(* PLC project Senza_nome, Sconosciuto Senza_nome 1 *)
(* stored: creationDateTime 2020-04-13T10:39:50, modificationDateTime 2020-06-24T12:04:16 *)

FUNCTION_BLOCK genera
  VAR_INPUT
    generate : BOOL;  (* generazione di un nuovo veicolo all'ingresso *)
  END_VAR
  VAR
    veicoli : ARRAY[1..10] OF INT;
    current_array_pos : INT := 1;
  END_VAR
  VAR_OUTPUT
    weight : INT;  (* peso "rilevato" *)
  END_VAR

            (* Blocco che simula l'ingresso di veicoli di differente peso*)
(* peso<=250= moto, peso>250 & peso <900= auto, peso>=900=camion*)

(* Definizione valori array di prova*)
veicoli[1] := 100;
veicoli[2] := 1454;
veicoli[3] := 807;
veicoli[4] := 252;
veicoli[5] := 1068;
veicoli[6] := 908;
veicoli[7] := 309;
veicoli[8] := 154;
veicoli[9] := 603;
veicoli[10] := 414;

if (generate=TRUE) then
  weight := veicoli[current_array_pos];
end_if;

current_array_pos := current_array_pos + 1;

(* Evito overflow array*)
if current_array_pos > 10 then
  current_array_pos := 1;
end_if;



          
END_FUNCTION_BLOCK

FUNCTION_BLOCK exit_sel
  VAR_INPUT
    confirm : BOOL := 0;  (* conferma veicolo in uscita *)
    slct : BOOL := 0;  (* selezione veicolo in uscita *)
  END_VAR
  VAR_OUTPUT
    veicolo : REAL;  (* veicolo selezionato *)
  END_VAR
  VAR
    auto : REAL := 1.0;
    moto : REAL := 0.50;
    camion : REAL := 2.0;
  END_VAR
  VAR_OUTPUT
    apri_sbarra : BOOL := 0;  (* abilitazione della sbarra d'uscita al piano *)
    cat : STRING;  (* uscita a monitor del tipo di veicolo in uscita *)
  END_VAR
  VAR
    tipo : INT;  (* tipologia di veicolo in uscita *)
    R_TRIG0 : R_TRIG;
  END_VAR

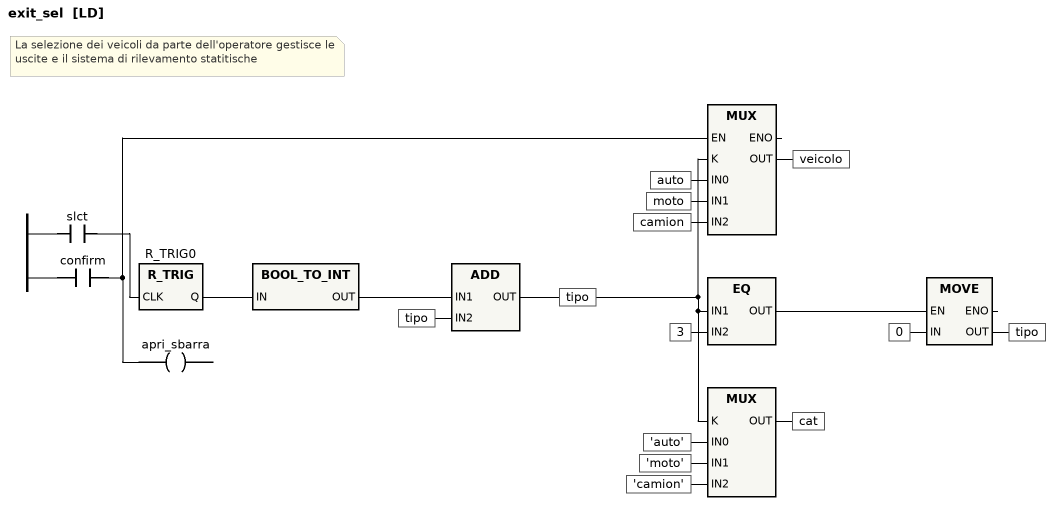
(* LD diagram, written out as Structured Text *)
IF confirm THEN veicolo := MUX(tipo, auto, moto, camion); END_IF;
apri_sbarra := confirm;
R_TRIG0(CLK := slct);
tipo := BOOL_TO_INT(R_TRIG0.Q) + tipo;
cat := MUX(tipo, 'auto', 'moto', 'camion');
(* La selezione dei veicoli da parte dell'operatore gestisce le uscite e il sistema di rilevamento statitische *)
IF tipo = 3 THEN tipo := 0; END_IF;
END_FUNCTION_BLOCK

FUNCTION_BLOCK gettoniera
  VAR_INPUT
    enable : BOOL := 0;  (* abilitazione/disabilitazione pagamento *)
    euro_1 : BOOL := 0;  (* rileva l'inserimento di 1€ *)
    euro_2 : BOOL := 0;  (* rileva l'inserimento di 2€ *)
    euro_50c : BOOL := 0;  (* rileva l'inserimento di 0.50€ *)
    ore : BOOL := 0;  (* ore di permanenza nel parcheggio *)
    tariffa : REAL := 1.0;  (* tariffa applicata in base al tipo di veicolo *)
  END_VAR
  VAR
    tot : REAL := 0.0;  (* totale inserito dall'utente *)
    prc : REAL := 1.0;
  END_VAR
  VAR_OUTPUT
    prezzo : REAL := 1.0;  (* uscita a schermo prezzo parcheggio *)
    tot_mon : REAL := 0.0;  (* uscita a schermo totale inserito *)
    hrs : INT := 0;  (* uscita a schermo ore *)
  END_VAR
  VAR
    ora : INT := 1;  (* conteggio delle ore *)
  END_VAR
  VAR_OUTPUT
    apri_sbarra : BOOL := 0;  (* apertura della sbarra dopo il pagamento *)
  END_VAR
  VAR
    R_TRIG0 : R_TRIG;
    R_TRIG1 : R_TRIG;
  END_VAR
  VAR_OUTPUT
    resto : REAL := 0.0;  (* resto erogato *)
  END_VAR
  VAR
    R_TRIG2 : R_TRIG;
    R_TRIG3 : R_TRIG;
    R_TRIG4 : R_TRIG;
    CTUD0 : CTUD;
  END_VAR
  VAR  (* added by the conversion: wires and edge detectors of the diagram *)
    R_TRIG1_2 : R_TRIG;
    _ADD185_OUT : REAL;
    _GE14_ENO : BOOL;
    _GE14_OUT : BOOL;
    R_TRIG2_2 : R_TRIG;
    _ADD16_ENO : BOOL;
    _ADD16_OUT : REAL;
    R_TRIG3_2 : R_TRIG;
    _SUB171_ENO : BOOL;
    _SUB171_OUT : REAL;
    _MOVE134_ENO : BOOL;
    _MOVE134_OUT : REAL;
    _LIMIT200_OUT : INT;
    _BOOL_TO_INT161_ENO : BOOL;
    _BOOL_TO_INT161_OUT : INT;
  END_VAR

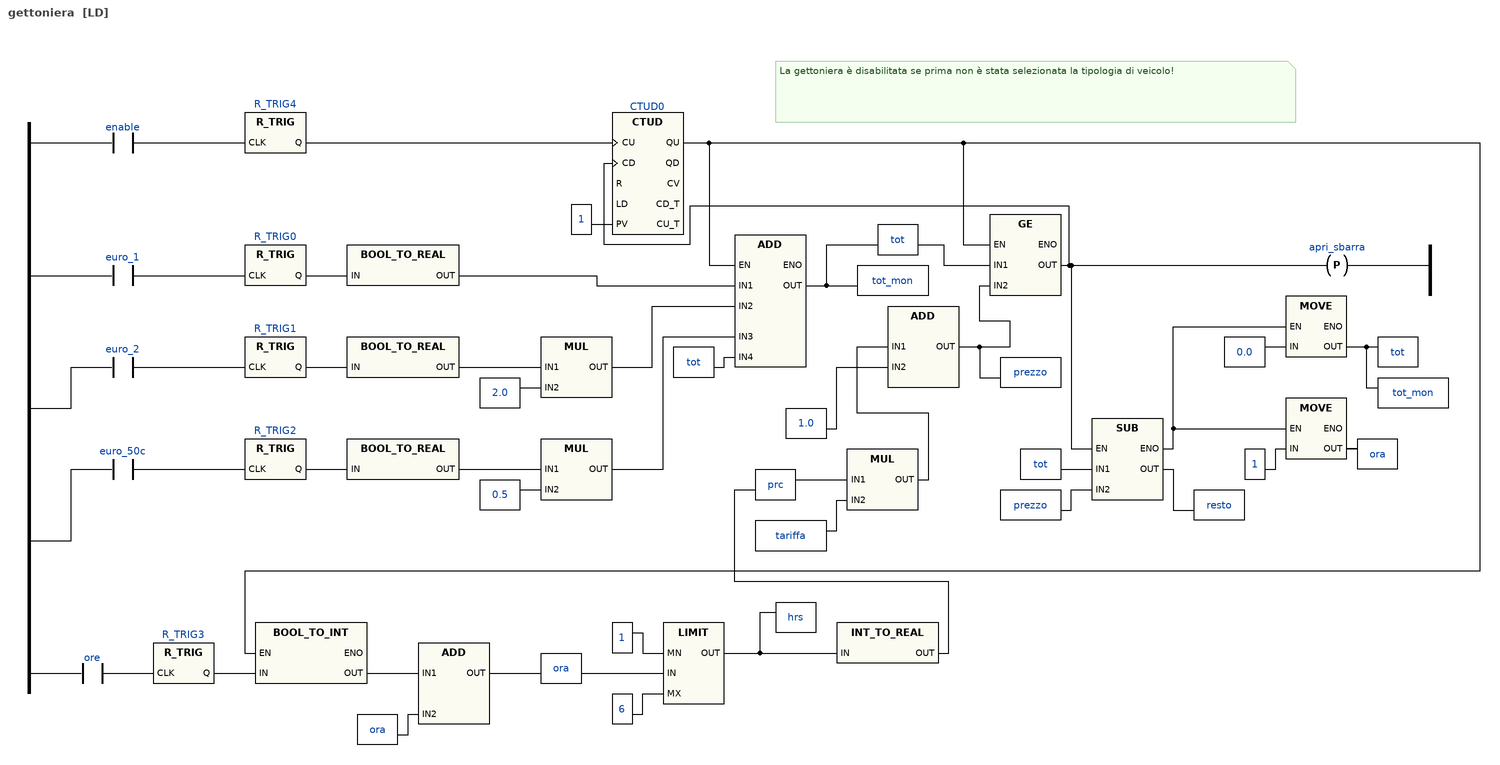
(* LD diagram, written out as Structured Text *)
(* La gettoniera è disabilitata se prima non è stata selezionata la tipologia di veicolo! *)
R_TRIG4(CLK := enable);
R_TRIG1_2(CLK := R_TRIG4.Q);
_ADD185_OUT := prc * tariffa + 1.0;
_GE14_OUT := GE(EN := CTUD0.QU, IN1 := tot, IN2 := _ADD185_OUT, ENO => _GE14_ENO);
R_TRIG2_2(CLK := _GE14_OUT);
CTUD0(CU := R_TRIG1_2.Q, CD := R_TRIG2_2.Q, PV := 1);
R_TRIG0(CLK := euro_1);
R_TRIG1(CLK := euro_2);
R_TRIG2(CLK := euro_50c);
_ADD16_OUT := ADD(EN := CTUD0.QU, IN1 := BOOL_TO_REAL(R_TRIG0.Q), IN2 := BOOL_TO_REAL(R_TRIG1.Q) * 2.0, IN3 := BOOL_TO_REAL(R_TRIG2.Q) * 0.5, IN4 := tot, ENO => _ADD16_ENO);
IF _ADD16_ENO THEN tot := _ADD16_OUT; END_IF;
R_TRIG3_2(CLK := _GE14_OUT);
apri_sbarra := R_TRIG3_2.Q;
IF _ADD16_ENO THEN tot_mon := _ADD16_OUT; END_IF;
_SUB171_OUT := SUB(EN := _GE14_OUT, IN1 := tot, IN2 := prezzo, ENO => _SUB171_ENO);
_MOVE134_OUT := MOVE(EN := _SUB171_ENO, IN := 0.0, ENO => _MOVE134_ENO);
IF _MOVE134_ENO THEN tot := _MOVE134_OUT; END_IF;
prezzo := _ADD185_OUT;
IF _MOVE134_ENO THEN tot_mon := _MOVE134_OUT; END_IF;
IF _SUB171_ENO THEN ora := 1; END_IF;
_LIMIT200_OUT := LIMIT(1, ora, 6);
prc := INT_TO_REAL(_LIMIT200_OUT);
IF _SUB171_ENO THEN resto := _SUB171_OUT; END_IF;
hrs := _LIMIT200_OUT;
R_TRIG3(CLK := ore);
_BOOL_TO_INT161_OUT := BOOL_TO_INT(EN := CTUD0.QU, IN := R_TRIG3.Q, ENO => _BOOL_TO_INT161_ENO);
ora := _BOOL_TO_INT161_OUT + ora;
END_FUNCTION_BLOCK

FUNCTION_BLOCK park_stats
  VAR_INPUT
    en_calc : BOOL := 0;  (* abilitazione del conteggio dei ricavi *)
    guad : REAL;  (* pedaggio riscosso *)
    tot_auto1 : INT;  (* totale auto presenti piano terra *)
    tot_moto1 : INT;  (* totale moto presenti piano terra *)
    tot_camion1 : INT;  (* totale camion presenti piano terra *)
    tot_auto2 : INT;  (* totale auto presenti primo piano *)
    tot_moto2 : INT;  (* totale moto presenti primo piano *)
    tot_camion2 : INT;  (* totale camion presenti primo piano *)
  END_VAR
  VAR_OUTPUT
    tot_auto : INT := 0;  (* auto presenti nell'intero parcheggio *)
    tot_moto : INT := 0;  (* moto presenti nell'intero parcheggio *)
    tot_camion : INT := 0;  (* camion presenti nell'intero parcheggio *)
    incasso : REAL := 0.0;  (* incasso giornaliero *)
    daily_vhcl : INT := 0;  (* totale dei veicoli che hanno transitato in un giorno *)
  END_VAR
  VAR
    R_TRIG0 : R_TRIG;
  END_VAR

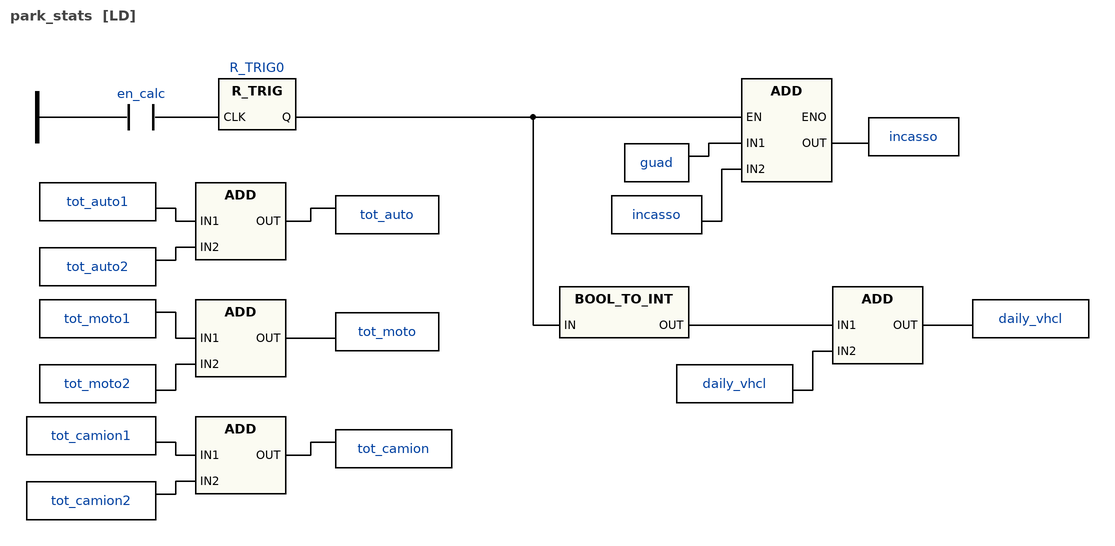
(* LD diagram, written out as Structured Text *)
R_TRIG0(CLK := en_calc);
IF R_TRIG0.Q THEN incasso := guad + incasso; END_IF;
tot_auto := tot_auto1 + tot_auto2;
daily_vhcl := BOOL_TO_INT(R_TRIG0.Q) + daily_vhcl;
tot_moto := tot_moto1 + tot_moto2;
tot_camion := tot_camion1 + tot_camion2;
END_FUNCTION_BLOCK

FUNCTION_BLOCK vehicle_cnt
  VAR_INPUT
    confirm_enter : BOOL := 0;  (* abilitazione per i contatori di incremento per un tipo di veicolo *)
    confirm_exit : BOOL := 0;  (* abilitazione per i contatori di decremento per un tipo di veicolo *)
    veicolo_in : REAL;  (* tipologia di veicolo in ingresso *)
    veicolo_out : REAL;  (* tipologia di veicolo in uscita *)
  END_VAR
  VAR_OUTPUT
    tot_auto : INT := 0;  (* totale auto presenti nel piano *)
    tot_moto : INT := 0;  (* totale moto presenti nel piano *)
    tot_camion : INT := 0;  (* totale camion presenti nel piano *)
  END_VAR
  VAR
    cap : INT := 4;  (* capacità di conteggio (legata al numero di veicoli per piano) *)
    R_TRIG0 : R_TRIG;
    CTUD0 : CTUD;
    CTUD1 : CTUD;
    CTUD2 : CTUD;
    R_TRIG1 : R_TRIG;
  END_VAR
  VAR  (* added by the conversion: wires and edge detectors of the diagram *)
    _EQ13_ENO : BOOL;
    _EQ13_OUT : BOOL;
    R_TRIG1_2 : R_TRIG;
    _EQ26_ENO : BOOL;
    _EQ26_OUT : BOOL;
    R_TRIG2 : R_TRIG;
    _EQ10_ENO : BOOL;
    _EQ10_OUT : BOOL;
    R_TRIG3 : R_TRIG;
    _EQ23_ENO : BOOL;
    _EQ23_OUT : BOOL;
    R_TRIG4 : R_TRIG;
    _EQ14_ENO : BOOL;
    _EQ14_OUT : BOOL;
    R_TRIG5 : R_TRIG;
    _EQ27_ENO : BOOL;
    _EQ27_OUT : BOOL;
    R_TRIG6 : R_TRIG;
  END_VAR

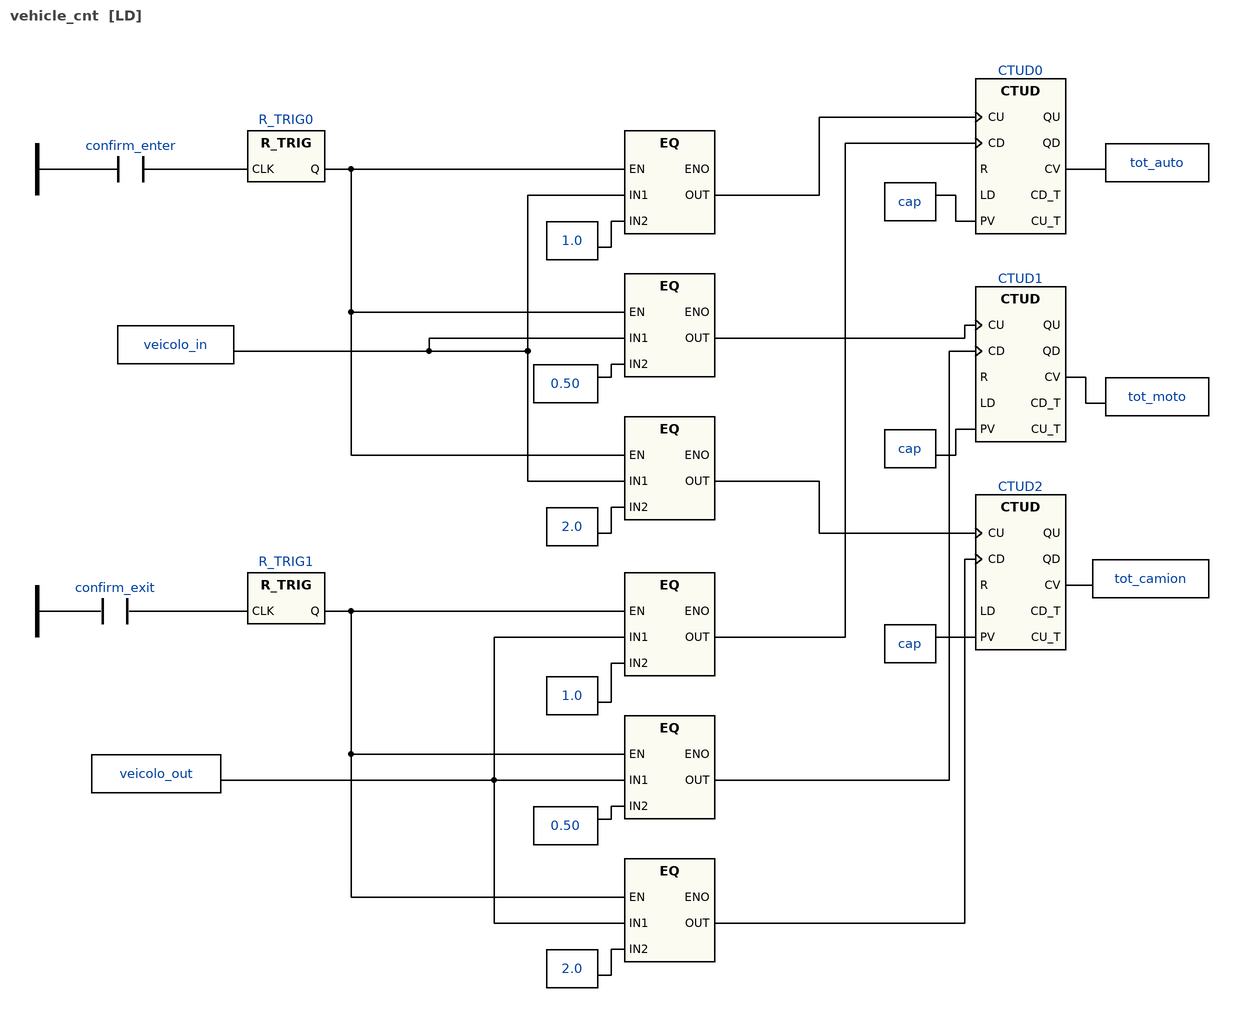
(* LD diagram, written out as Structured Text *)
R_TRIG0(CLK := confirm_enter);
_EQ13_OUT := EQ(EN := R_TRIG0.Q, IN1 := veicolo_in, IN2 := 1.0, ENO => _EQ13_ENO);
R_TRIG1_2(CLK := _EQ13_OUT);
R_TRIG1(CLK := confirm_exit);
_EQ26_OUT := EQ(EN := R_TRIG1.Q, IN1 := veicolo_out, IN2 := 1.0, ENO => _EQ26_ENO);
R_TRIG2(CLK := _EQ26_OUT);
CTUD0(CU := R_TRIG1_2.Q, CD := R_TRIG2.Q, PV := cap);
tot_auto := CTUD0.CV;
_EQ10_OUT := EQ(EN := R_TRIG0.Q, IN1 := veicolo_in, IN2 := 0.50, ENO => _EQ10_ENO);
R_TRIG3(CLK := _EQ10_OUT);
_EQ23_OUT := EQ(EN := R_TRIG1.Q, IN1 := veicolo_out, IN2 := 0.50, ENO => _EQ23_ENO);
R_TRIG4(CLK := _EQ23_OUT);
CTUD1(CU := R_TRIG3.Q, CD := R_TRIG4.Q, PV := cap);
tot_moto := CTUD1.CV;
_EQ14_OUT := EQ(EN := R_TRIG0.Q, IN1 := veicolo_in, IN2 := 2.0, ENO => _EQ14_ENO);
R_TRIG5(CLK := _EQ14_OUT);
_EQ27_OUT := EQ(EN := R_TRIG1.Q, IN1 := veicolo_out, IN2 := 2.0, ENO => _EQ27_ENO);
R_TRIG6(CLK := _EQ27_OUT);
CTUD2(CU := R_TRIG5.Q, CD := R_TRIG6.Q, PV := cap);
tot_camion := CTUD2.CV;
END_FUNCTION_BLOCK

FUNCTION_BLOCK vehicle_sel
  VAR_INPUT
    invio : BOOL := 0;  (* conferma scelta *)
    slct : BOOL := 0;  (* selezionatore (se >2 torna a 0) *)
    weight : INT;  (* rilevatore del peso del veicolo in ingresso *)
  END_VAR
  VAR_OUTPUT
    abilita : BOOL;  (* abilitazione gettoniera *)
    cat : STRING;  (* uscita a schermo *)
  END_VAR
  VAR
    veicleDetect : INT;  (* veicolo determinato in base al peso *)
  END_VAR
  VAR_OUTPUT
    veicolo : REAL := 1.0;  (* veicolo selezionato *)
  END_VAR
  VAR
    tipo : INT := 0;  (* auto=0, moto=1,camion=2 *)
    auto : REAL := 1.0;  (* tariffa auto *)
    moto : REAL := 0.50;  (* tariffa moto *)
    camion : REAL := 2.00;  (* tariffa camion *)
    R_TRIG0 : R_TRIG;
  END_VAR
  VAR  (* added by the conversion: wires and edge detectors of the diagram *)
    _AND61_OUT : BOOL;
    _AND44_OUT : BOOL;
    _GT47_OUT : BOOL;
    _EQ56_ENO : BOOL;
    _EQ56_OUT : BOOL;
    _MUX1_ENO : BOOL;
    _MUX1_OUT : REAL;
  END_VAR

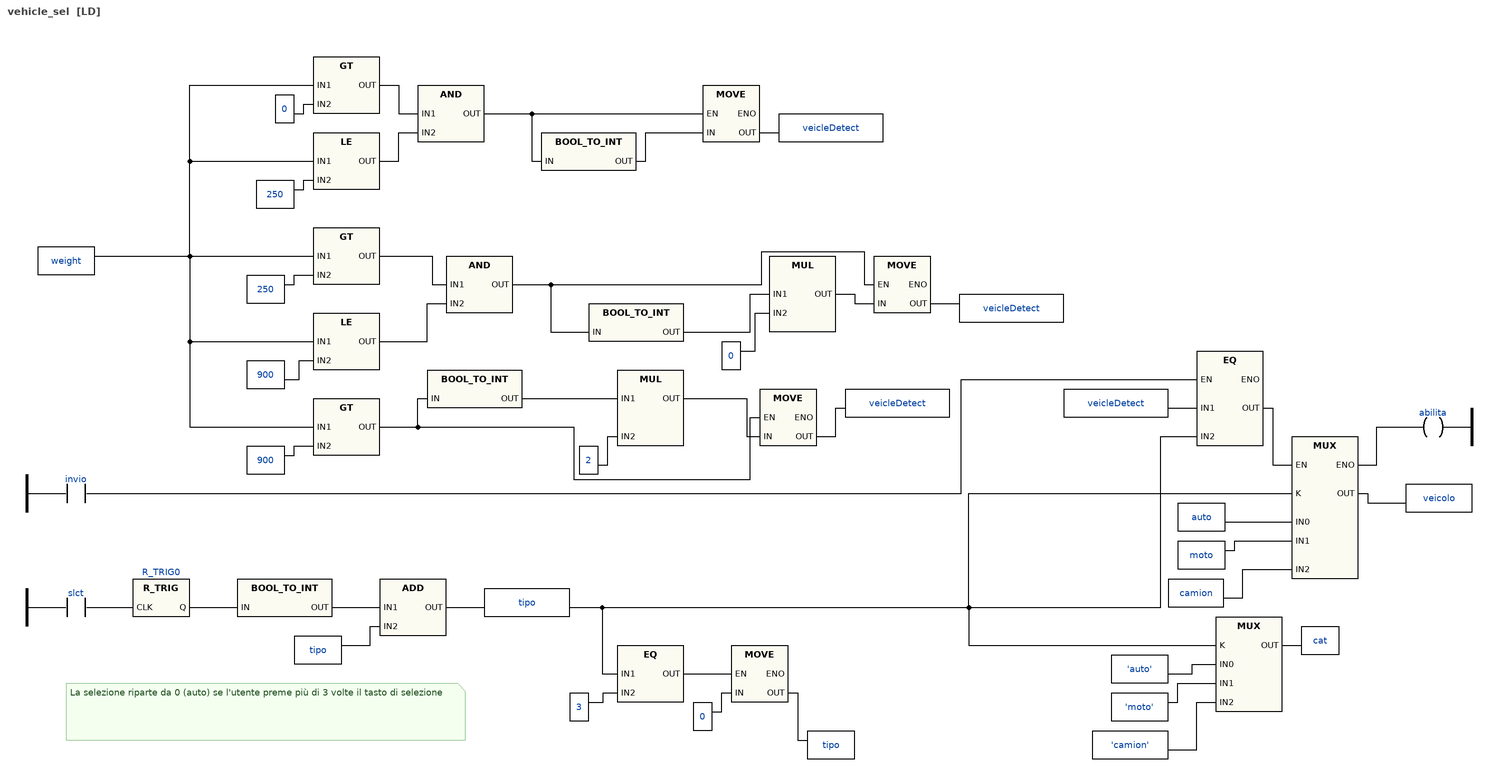
(* LD diagram, written out as Structured Text *)
_AND61_OUT := weight > 0 AND weight <= 250;
IF _AND61_OUT THEN veicleDetect := BOOL_TO_INT(_AND61_OUT); END_IF;
_AND44_OUT := weight > 250 AND weight <= 900;
IF _AND44_OUT THEN veicleDetect := BOOL_TO_INT(_AND44_OUT) * 0; END_IF;
_GT47_OUT := weight > 900;
IF _GT47_OUT THEN veicleDetect := BOOL_TO_INT(_GT47_OUT) * 2; END_IF;
_EQ56_OUT := EQ(EN := invio, IN1 := veicleDetect, IN2 := tipo, ENO => _EQ56_ENO);
_MUX1_OUT := MUX(EN := _EQ56_OUT, K := tipo, IN0 := auto, IN1 := moto, IN2 := camion, ENO => _MUX1_ENO);
abilita := _MUX1_ENO;
IF _MUX1_ENO THEN veicolo := _MUX1_OUT; END_IF;
R_TRIG0(CLK := slct);
tipo := BOOL_TO_INT(R_TRIG0.Q) + tipo;
cat := MUX(tipo, 'auto', 'moto', 'camion');
(* La selezione riparte da 0 (auto) se l'utente preme più di 3 volte il tasto di selezione *)
IF tipo = 3 THEN tipo := 0; END_IF;
END_FUNCTION_BLOCK

PROGRAM parking
  VAR
    start : BOOL := 0;  (* inizializzazione parcheggio *)
  END_VAR
  VAR_INPUT
    gen : BOOL := 0;  (* generazione veicolo *)
  END_VAR
  VAR
    slct : BOOL := 0;  (* selezione del tipo di veicolo (0 auto, 1 moto, 3 camion) *)
  END_VAR
  VAR_INPUT
    conferma : BOOL := 0;  (* conferma selezione veicolo *)
    cent_50 : BOOL := 0;  (* inserimento moneta €0,50 *)
    euro_1 : BOOL := 0;  (* inserimento moneta €1 *)
    euro_2 : BOOL := 0;  (* inserimento moneta €2 *)
    ora : BOOL := 0;  (* selezione delle ore (max 6) *)
    slct_exit1 : BOOL := 0;  (* selettore veicolo in uscita piano terra *)
    slct_exit2 : BOOL := 0;  (* selettore veicolo in uscita primo piano *)
    conf1 : BOOL := 0;  (* conferma uscita piano terra *)
    conf2 : BOOL := 0;  (* conferma uscita primo piano *)
  END_VAR
  VAR_OUTPUT
    resto : REAL := 0.0;  (* resto *)
    prezzo : REAL := 0.0;  (* prezzo da pagare *)
  END_VAR
  VAR
    stop : BOOL := 0;  (* chiusura parcheggio *)
    cap : INT := 4;  (* capienza di ogni piano *)
    sbarra1 : BOOL := 0;  (* sbarra d'ingresso piano terra *)
    sbarra2 : BOOL := 0;  (* sbarra d'ingresso primo piano *)
  END_VAR
  VAR_INPUT
    sbarra1_man : BOOL := 0;  (* pulsante di attivazione manuale della sbarra all'ingresso del piano 1 *)
    sbarra2_man : BOOL := 0;  (* pulsante di attivazione manuale della sbarra all'ingresso del secondo piano *)
  END_VAR
  VAR
    enter_1 : BOOL := 0;  (* apertura primo ingresso *)
    piano1_full : BOOL := 0;  (* segnalazione capienza max raggiunta piano terra *)
    piano2_full : BOOL := 0;  (* segnalazione capienza max raggiunta primo piano *)
    exit_1 : BOOL := 0;  (* uscita primo piano *)
  END_VAR
  VAR_OUTPUT
    exit_2 : BOOL := 0;  (* uscita secondo piano *)
    enter_2 : BOOL := 0;  (* apertura secondo ingresso *)
    park_full : BOOL := 0;  (* garage totalmente pieno *)
  END_VAR
  VAR
    TON0 : TON;  (* abilitazione entrata primo piano *)
  END_VAR
  VAR_INPUT
    temp1 : TIME := T#2s;  (* tempo apertura ingresso1 *)
    temp2 : TIME := T#4s;  (* tempo apertura ingresso2 *)
    temp3 : TIME := T#1s;  (* tempo apertura ingresso2 *)
  END_VAR
  VAR
    CTUD0 : CTUD;  (* contatore auto primo piano *)
    exit1_en : BOOL := 0;  (* uscita primo piano *)
    exit2_en : BOOL := 0;  (* uscita secondo piano *)
    TON1 : TON;  (* abilitazione uscita primo piano *)
    TON2 : TON;  (* abilitazione ingresso secondo piano *)
    CTUD1 : CTUD;  (* contatore auto secondo piano *)
    TON3 : TON;  (* abilitazione uscita secondo piano *)
    TOF1 : TOF;  (* segnalazione posto disponibile al secondo piano *)
    gettoniera0 : gettoniera;  (* contamonete (con resto) *)
    vehicle_sel0 : vehicle_sel;  (* selettore del tipo di veicolo *)
    vehicle_cnt0 : vehicle_cnt;
    exit_sel0 : exit_sel;
    vehicle_cnt1 : vehicle_cnt;
    exit_sel1 : exit_sel;
    park_stats0 : park_stats;
    genera0 : genera;
    R_TRIG0 : R_TRIG;
  END_VAR
  VAR  (* added by the conversion: wires and edge detectors of the diagram *)
    R_TRIG1 : R_TRIG;
    R_TRIG2 : R_TRIG;
    R_TRIG3 : R_TRIG;
    R_TRIG4 : R_TRIG;
  END_VAR

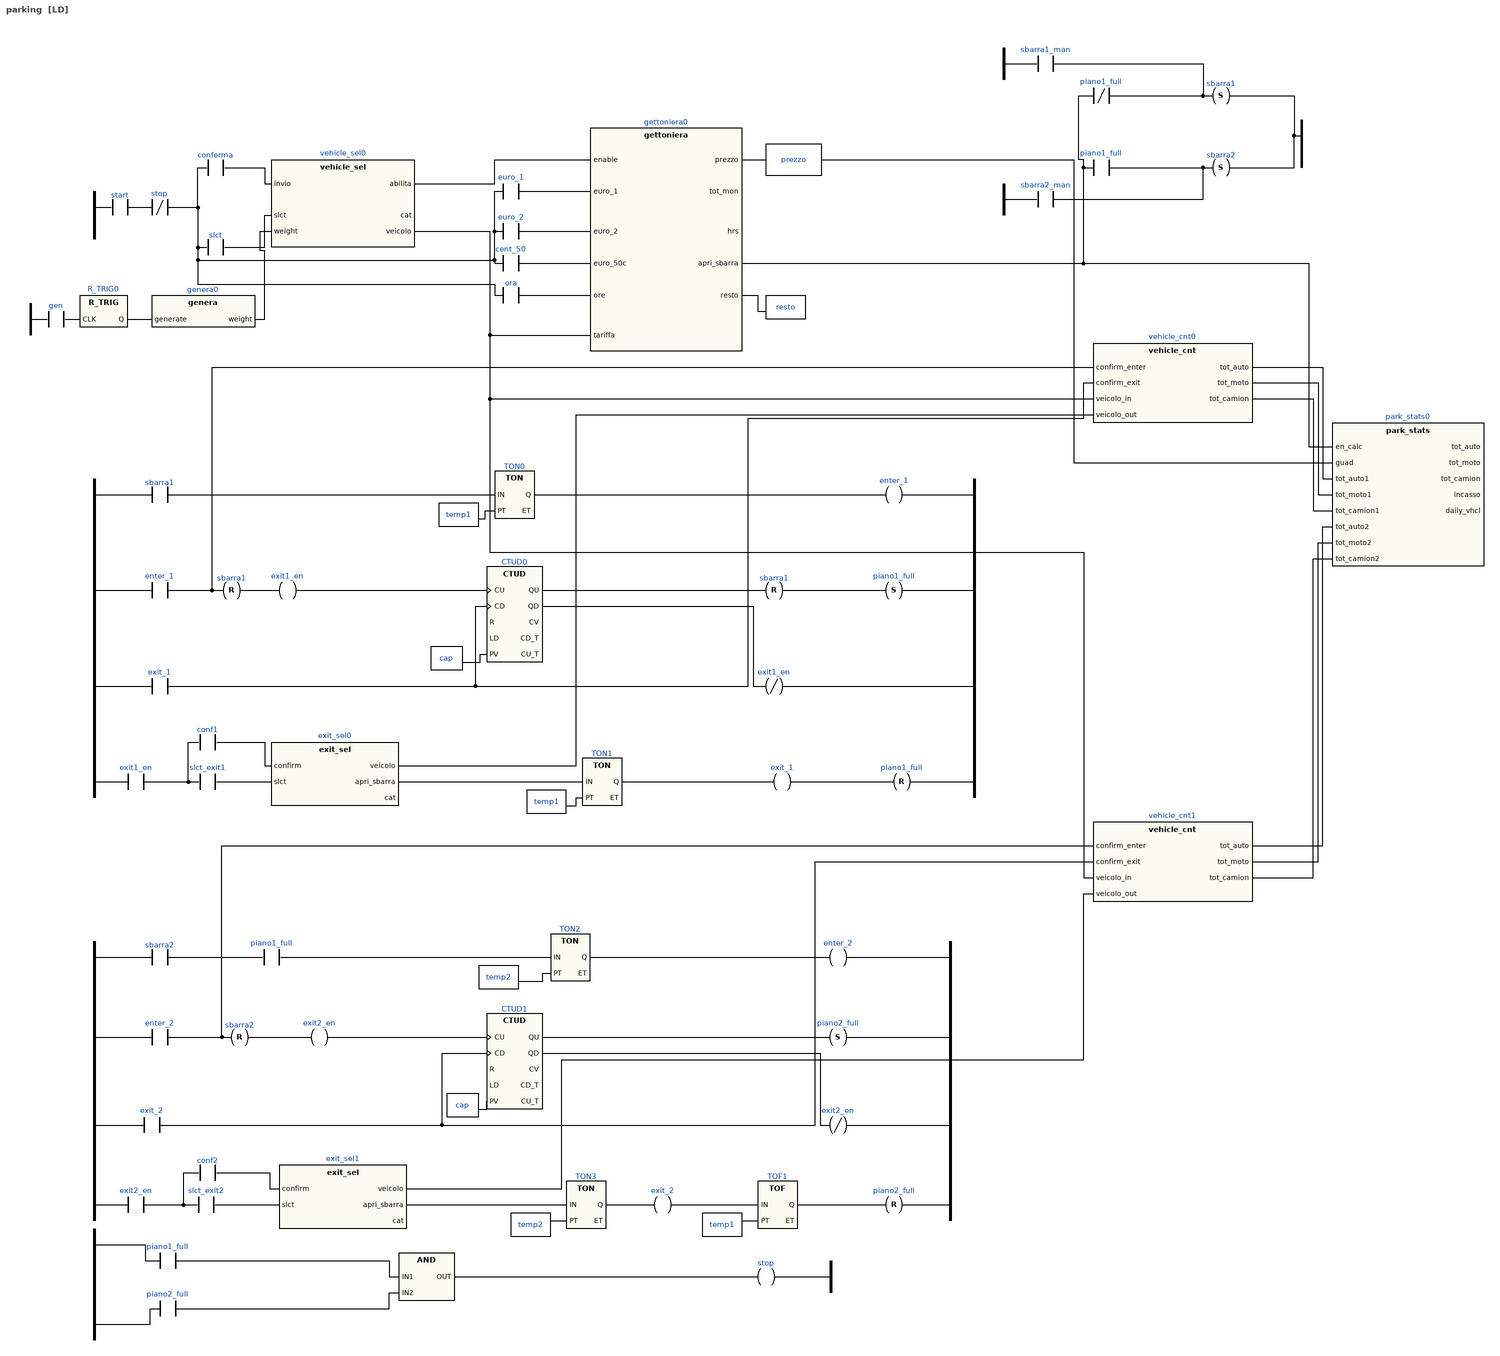
(* LD diagram, written out as Structured Text *)
R_TRIG0(CLK := gen);
genera0(generate := R_TRIG0.Q);
vehicle_sel0(invio := start AND NOT stop AND conferma, slct := start AND NOT stop AND slct, weight := genera0.weight);
gettoniera0(enable := vehicle_sel0.abilita, euro_1 := start AND NOT stop AND euro_1, euro_2 := start AND NOT stop AND euro_2, euro_50c := start AND NOT stop AND cent_50, ore := start AND NOT stop AND ora, tariffa := vehicle_sel0.veicolo);
IF gettoniera0.apri_sbarra AND NOT piano1_full OR sbarra1_man THEN sbarra1 := TRUE; END_IF;
prezzo := gettoniera0.prezzo;
IF gettoniera0.apri_sbarra AND piano1_full OR sbarra2_man THEN sbarra2 := TRUE; END_IF;
resto := gettoniera0.resto;
TON0(IN := sbarra1, PT := temp1);
enter_1 := TON0.Q;
IF enter_1 THEN sbarra1 := FALSE; END_IF;
exit1_en := enter_1;
R_TRIG1(CLK := enter_1);
R_TRIG2(CLK := exit_1);
CTUD0(CU := R_TRIG1.Q, CD := R_TRIG2.Q, PV := cap);
IF CTUD0.QU THEN sbarra1 := FALSE; END_IF;
IF CTUD0.QU THEN piano1_full := TRUE; END_IF;
exit1_en := NOT CTUD0.QD;
exit_sel0(confirm := exit1_en AND conf1, slct := exit1_en AND slct_exit1);
TON1(IN := exit_sel0.apri_sbarra, PT := temp1);
exit_1 := TON1.Q;
IF TON1.Q THEN piano1_full := FALSE; END_IF;
TON2(IN := sbarra2 AND piano1_full, PT := temp2);
enter_2 := TON2.Q;
IF enter_2 THEN sbarra2 := FALSE; END_IF;
exit2_en := enter_2;
R_TRIG3(CLK := enter_2);
R_TRIG4(CLK := exit_2);
CTUD1(CU := R_TRIG3.Q, CD := R_TRIG4.Q, PV := cap);
IF CTUD1.QU THEN piano2_full := TRUE; END_IF;
exit2_en := NOT CTUD1.QD;
exit_sel1(confirm := exit2_en AND conf2, slct := exit2_en AND slct_exit2);
TON3(IN := exit_sel1.apri_sbarra, PT := temp2);
exit_2 := TON3.Q;
TOF1(IN := TON3.Q, PT := temp1);
IF TOF1.Q THEN piano2_full := FALSE; END_IF;
stop := piano1_full AND piano2_full;
vehicle_cnt0(confirm_enter := enter_1, confirm_exit := exit_1, veicolo_in := vehicle_sel0.veicolo, veicolo_out := exit_sel0.veicolo);
vehicle_cnt1(confirm_enter := enter_2, confirm_exit := exit_2, veicolo_in := vehicle_sel0.veicolo, veicolo_out := exit_sel1.veicolo);
park_stats0(en_calc := gettoniera0.apri_sbarra, guad := prezzo, tot_auto1 := vehicle_cnt0.tot_auto, tot_moto1 := vehicle_cnt0.tot_moto, tot_camion1 := vehicle_cnt0.tot_camion, tot_auto2 := vehicle_cnt1.tot_auto, tot_moto2 := vehicle_cnt1.tot_moto, tot_camion2 := vehicle_cnt1.tot_camion);
END_PROGRAM

CONFIGURATION Config0
  RESOURCE Res0 ON PLC
    TASK task0(INTERVAL := T#20ms, PRIORITY := 0);
    PROGRAM instance0 WITH task0 : parking;
  END_RESOURCE
END_CONFIGURATION
